PROGRAM MAIN
VAR
	Variable:BOOL;
END_VAR

END_PROGRAM

(* stored: Version 1.1.0.1, ProductVersion 3.1.4024.9
   POU MAIN: Id {73a60ecc-3bcd-4f0c-b1f9-4d748229b0f5}, SpecialFunc None *)
